# B&R Automation Studio project CleanChemi_SiteManagementSystem (part 4)

#### HA_Find_R.st
```iecst
(* Returns Right index of substring. Negative values are Errors. *)
FUNCTION HA_Find_R
	IF pBuffer = 0 OR pSearch = 0 THEN
		HA_Find_R	 						:= -2;
	ELSE
		Internal.sB							:= brsstrlen(pBuffer);
		Internal.sS							:= brsstrlen(pSearch);
		IF Internal.sB = 0 OR Internal.sB < Internal.sS THEN
		HA_Find_R	 						:= -3;
		END_IF;
	END_IF;
	IF HA_Find_R = 0 THEN
		HA_Find_R							:= -1;
		IF Internal.sS = 0 THEN
			HA_Find_R 						:= 0;
			RETURN;
		ELSE
			FOR Internal.i := 0 TO Internal.sB-Internal.sS DO
				IF brsmemcmp(pBuffer+Internal.i,pSearch,Internal.sS) = 0 THEN
					HA_Find_R 				:= Internal.i+Internal.sS;
					RETURN;
				END_IF;
			END_FOR;
		END_IF;
	END_IF;
END_FUNCTION
```

#### HA_Find_Extract.st
```iecst
(* Negative values are Errors. *)
FUNCTION HA_Find_Extract
	IF pBuffer = 0 OR pSearchL = 0 OR pSearchR = 0 OR pExtractADR = 0 OR pExtractSIZEOF = 0 THEN
		HA_Find_Extract 						:= -2;
	ELSE
		Internal.sB								:= brsstrlen(pBuffer);
		Internal.sSL							:= brsstrlen(pSearchL);
		Internal.sSR							:= brsstrlen(pSearchR);
		IF Internal.sB = 0 OR Internal.sB < (Internal.sSL + Internal.sSR + 1) THEN
			HA_Find_Extract 					:= -3;
		END_IF;
	END_IF;
	IF HA_Find_Extract = 0 THEN
		HA_Find_Extract							:= -1;
		Internal.P1 							:= HA_Find_R(pBuffer,pSearchL);
		IF Internal.P1 >= 0 THEN
			Internal.P2 						:= HA_Find_L(pBuffer+Internal.P1,pSearchR);
			IF Internal.P2 >= 0 THEN
				Internal.Pos 					:= Internal.P1 + pBuffer;
				Internal.Len 					:= DINT_TO_UDINT(Internal.P2);
				brsmemcpy(pExtractADR,ADR(Internal.Pos),4);
				brsmemcpy(pExtractSIZEOF,ADR(Internal.Len),4);
				HA_Find_Extract					:= Internal.P1+Internal.P2+Internal.sSR;
			END_IF;
		END_IF;
	END_IF;
END_FUNCTION
```

### Library Logical/Libraries/API_Login (IEC)

#### Enums.typ
```iecst
TYPE
	LoginState_Enum :
		(
		IDLE_I,
		REQ_AUTH_C,
		REQ_AUTH_W,
		PARSE_AUTH_JSON_C,
		PARSE_AUTH_JSON_W,
		REQ_USER_INFO_W,
		REQ_USER_INFO_C,
		PARSE_USER_INFO_C,
		PARSE_USER_INFO_W,
		CREATE_USER_C,
		CREATE_USER_W,
		SET_PASSWORD_C,
		SET_PASSWORD_W,
		SET_ROLES_W,
		SET_ROLES_C,
		USER_CREATED_SUCCESSS,
		LOGIN_API_ERROR
		);
END_TYPE
```

#### API_Login.fun - Exported functions and function blocks
```iecst
FUNCTION_BLOCK API_Login_FB
	VAR_INPUT
		bExecute : BOOL;
		sUser : STRING[80];
		sPassword : STRING[80];
	END_VAR
	VAR_OUTPUT
		LoginState : LoginState_Enum;
		UserID : STRING[80];
		Password : STRING[80];
		Name : STRING[80];
		Error : BOOL;
		ErrorInfo : STRING[80];
		Done : BOOL;
		Authorization_Bearer : STRING[300];
		ReturnedLastName : STRING[80];
		ReturnedFirstName : STRING[80];
		ReturnedID : UINT;
		ReturnedRole : STRING[80];
	END_VAR
	VAR_IN_OUT
		RequestHeader : httpRequestHeader_t;
		HttpClientRef : httpsClient;
	END_VAR
	VAR
		IdxJSON : DINT;
		GET_UserInfo : GET_UserInfo_FB;
		POST_Login : POST_Login_FB;
		HA_JSON_Parse : HA_JSON_Parse;
		ArUserAssignRole : ArUserAssignRole;
		ArUserSetPassword : ArUserSetPassword;
		JSON_Parsed : ARRAY[0..MAX_JSON_PARSE_PAIR_IDX] OF HA_JSON_Parse_Pair_typ;
		ArUserCreate : ArUserCreate;
	END_VAR
END_FUNCTION_BLOCK

{REDUND_ERROR} FUNCTION_BLOCK POST_Login_FB (*TODO: Add your comment here*) (*$GROUP=User,$CAT=User,$GROUPICON=User.png,$CATICON=User.png*)
	VAR_INPUT
		username : STRING[80];
		password : STRING[80];
		bEnable : BOOL;
		bRequest : BOOL;
	END_VAR
	VAR_OUTPUT
		Phase : UINT;
		Status : {REDUND_UNREPLICABLE} UINT;
		ResponseStatus : {REDUND_UNREPLICABLE} STRING[280];
		Authorization : STRING[200];
		ResponseData : {REDUND_UNREPLICABLE} STRING[2000];
	END_VAR
	VAR_IN_OUT
		HttpClientRef : httpsClient;
		RequestHeader : httpRequestHeader_t;
	END_VAR
	VAR
		Host : {REDUND_UNREPLICABLE} STRING[80];
		ResponseHeader : {REDUND_UNREPLICABLE} httpResponseHeader_t;
		Ressource : {REDUND_UNREPLICABLE} STRING[80];
		sHeader : {REDUND_UNREPLICABLE} STRING[300];
		bEnabled : {REDUND_UNREPLICABLE} BOOL;
		RequestDataJson : {REDUND_UNREPLICABLE} STRING[1000];
	END_VAR
END_FUNCTION_BLOCK

{REDUND_ERROR} FUNCTION_BLOCK GET_UserInfo_FB (*TODO: Add your comment here*) (*$GROUP=User,$CAT=User,$GROUPICON=User.png,$CATICON=User.png*)
	VAR_INPUT
		sAuthorization : STRING[250];
		bEnable : BOOL;
		bRequest : BOOL;
	END_VAR
	VAR_OUTPUT
		Phase : UINT;
		Status : {REDUND_UNREPLICABLE} UINT;
		ResponseStatus : {REDUND_UNREPLICABLE} STRING[280];
		ResponseData : {REDUND_UNREPLICABLE} STRING[2000];
	END_VAR
	VAR_IN_OUT
		HttpClientRef : httpsClient;
		RequestHeader : httpRequestHeader_t;
	END_VAR
	VAR
		Host : {REDUND_UNREPLICABLE} STRING[80];
		ResponseHeader : {REDUND_UNREPLICABLE} httpResponseHeader_t;
		Ressource : {REDUND_UNREPLICABLE} STRING[80];
		sHeader : {REDUND_UNREPLICABLE} STRING[400];
		bEnabled : {REDUND_UNREPLICABLE} BOOL;
		RequestDataJson : {REDUND_UNREPLICABLE} STRING[1000];
	END_VAR
END_FUNCTION_BLOCK
```

#### POST_Login.st
```iecst
(* TODO: Add your comment here *)
FUNCTION_BLOCK POST_Login_FB

	IF bEnable AND NOT bEnabled THEN
		bEnabled	:= TRUE;
		Ressource	:= '/auth/jwt/create/';
		RequestDataJson := CONCAT('{"username":"',username);
		RequestDataJson := CONCAT(	RequestDataJson,'","password":"');
		RequestDataJson := CONCAT(	RequestDataJson,password);
		RequestDataJson := CONCAT(	RequestDataJson,'"}');

		HttpClientRef.method 			:= httpMETHOD_POST;
		HttpClientRef.pUri 				:= ADR(Ressource);
		HttpClientRef.pRequestHeader	:= ADR(RequestHeader);
		HttpClientRef.pRequestData		:= ADR(RequestDataJson);
		HttpClientRef.requestDataLen	:= LEN(RequestDataJson)+2; //According to WireShark there is a /r/n in the packet that is not being accounted for which requires us to add 2 bytes to the length
		HttpClientRef.pResponseHeader	:= ADR(ResponseHeader);
		HttpClientRef.pResponseData 	:= ADR(ResponseData);
		HttpClientRef.responseDataSize	:= SIZEOF(ResponseData);

		RequestHeader.protocol			:= 'HTTP/1.1';
		RequestHeader.host				:= Host;
		RequestHeader.contentType		:= 'application/json';
		RequestHeader.contentLength		:=  LEN(RequestDataJson)+2; //According to WireShark there is a /r/n in the packet that is not being accounted for which requires us to add 2 bytes to the length
		RequestHeader.connection		:= 'keep-alive';
		RequestHeader.rawHeader.dataLen	:= LEN(sHeader);
		RequestHeader.rawHeader.pData	:= ADR(sHeader);

	ELSIF bEnable AND bEnabled THEN
		HttpClientRef.enable	:= TRUE;
		IF bRequest THEN
			HttpClientRef.send	:= TRUE;
		END_IF
	ELSIF NOT bEnable AND bEnabled THEN
		bEnabled	:= FALSE;
		bRequest	:= FALSE;
		HttpClientRef.enable	:= FALSE;
		HttpClientRef.send	:= FALSE;
	END_IF

	HttpClientRef();

	Status := HttpClientRef.status;
	Phase := HttpClientRef.phase;
	ResponseStatus := ResponseHeader.status;

END_FUNCTION_BLOCK
```

#### GET_UserInfo.st
```iecst
(* TODO: Add your comment here *)
FUNCTION_BLOCK GET_UserInfo_FB

	IF bEnable AND NOT bEnabled THEN
		bEnabled	:= TRUE;
		sHeader		:= CONCAT('Authorization: Bearer ',sAuthorization);
		Ressource	:= '/auth/users/me/';

		HttpClientRef.option 			:= httpOPTION_HTTP_11;
		HttpClientRef.method 			:= httpMETHOD_GET;
		HttpClientRef.pUri 				:= ADR(Ressource);
		HttpClientRef.pRequestHeader	:= ADR(RequestHeader);
		HttpClientRef.pRequestData		:= ADR(RequestDataJson);
		HttpClientRef.requestDataLen	:= LEN(RequestDataJson);
		HttpClientRef.pResponseHeader	:= ADR(ResponseHeader);
		HttpClientRef.pResponseData 	:= ADR(ResponseData);
		HttpClientRef.responseDataSize	:= SIZEOF(ResponseData);

		RequestHeader.protocol			:= 'HTTP/1.1';
		RequestHeader.contentType		:= 'application/json';
		RequestHeader.contentLength		:=  LEN(RequestDataJson);
		RequestHeader.connection		:= 'keep-alive';
		RequestHeader.rawHeader.dataLen	:= LEN(sHeader);
		RequestHeader.rawHeader.pData	:= ADR(sHeader);

	ELSIF bEnable AND bEnabled THEN
		HttpClientRef.enable	:= TRUE;
		IF bRequest THEN
			HttpClientRef.send	:= TRUE;
		END_IF
	ELSIF NOT bEnable AND bEnabled THEN
		bEnabled	:= FALSE;
		bRequest	:= FALSE;
		HttpClientRef.enable	:= FALSE;
		HttpClientRef.send	:= FALSE;
	END_IF

	HttpClientRef();

	Status := HttpClientRef.status;
	Phase := HttpClientRef.phase;
	ResponseStatus := ResponseHeader.status;

END_FUNCTION_BLOCK
```

#### API_Login_FB.st
```iecst
(* TODO: Add your comment here *)
FUNCTION_BLOCK API_Login_FB

	IF NOT bExecute THEN
		LoginState := IDLE_I;
	END_IF;

	CASE LoginState OF

		IDLE_I:

			GET_UserInfo.bEnable := FALSE;
			GET_UserInfo.bRequest := FALSE;
			POST_Login.bEnable := FALSE;
			POST_Login.bRequest := FALSE;
			HA_JSON_Parse.Enable := FALSE;
			ArUserSetPassword.Execute := FALSE;
			ArUserCreate.Execute := FALSE;
			brsmemset(ADR(Authorization_Bearer),0,SIZEOF(Authorization_Bearer));
			brsmemset(ADR(JSON_Parsed),0,SIZEOF(JSON_Parsed));
			ErrorInfo := '';

			Done := FALSE;
			Error := FALSE;

			IF bExecute THEN
				LoginState := REQ_AUTH_C;
			END_IF;

		REQ_AUTH_C:

			POST_Login.username := sUser;
			POST_Login.password := sPassword;

			POST_Login.bEnable := TRUE;
			POST_Login.bRequest := TRUE;

			LoginState := REQ_AUTH_W;

		REQ_AUTH_W:

			IF POST_Login.Status = 0 AND POST_Login.ResponseStatus = '200 OK' THEN
				LoginState := PARSE_AUTH_JSON_C;
			ELSIF  POST_Login.Status = 0 AND POST_Login.ResponseStatus = '401 Unauthorized' THEN
				LoginState := LOGIN_API_ERROR;
				ErrorInfo := POST_Login.ResponseStatus;
			ELSIF POST_Login.Status = 0 AND POST_Login.ResponseStatus = '400 Bad Request' THEN
				LoginState := LOGIN_API_ERROR;
				ErrorInfo := POST_Login.ResponseStatus;
			END_IF;

		PARSE_AUTH_JSON_C:

			POST_Login.bEnable := FALSE;
			POST_Login.bRequest := FALSE;
			HA_JSON_Parse.Enable := TRUE;
			HA_JSON_Parse.pBuffer := ADR(POST_Login.ResponseData);
			HA_JSON_Parse.pPairs := ADR(JSON_Parsed);

			LoginState := PARSE_AUTH_JSON_W;

		PARSE_AUTH_JSON_W:

			IF HA_JSON_Parse.Done THEN
				LoginState := REQ_USER_INFO_C;
			END_IF;

		REQ_USER_INFO_C:

			HA_JSON_Parse.Enable := FALSE;

			FOR IdxJSON := 0 TO MAX_JSON_PARSE_PAIR_IDX DO
				IF JSON_Parsed[IdxJSON].Name = 'access' THEN
					brsmemcpy(ADR(Authorization_Bearer),ADR(JSON_Parsed[IdxJSON].Value)+1,LEN(JSON_Parsed[IdxJSON].Value)-2);
					EXIT;
				END_IF;
			END_FOR;

			GET_UserInfo.bEnable := TRUE;
			GET_UserInfo.bRequest := TRUE;
			GET_UserInfo.sAuthorization := Authorization_Bearer;

			LoginState := REQ_USER_INFO_W;

		REQ_USER_INFO_W:

			IF GET_UserInfo.Status = 0 AND GET_UserInfo.ResponseStatus = '200 OK' THEN
				LoginState := PARSE_USER_INFO_C;
			ELSIF GET_UserInfo.Status = 0 AND GET_UserInfo.ResponseStatus = '401 Unauthorized' THEN
				LoginState := LOGIN_API_ERROR;
			END_IF;

		PARSE_USER_INFO_C:

			GET_UserInfo.bEnable := FALSE;
			GET_UserInfo.bRequest := FALSE;
			HA_JSON_Parse.Enable := TRUE;
			HA_JSON_Parse.pBuffer := ADR(GET_UserInfo.ResponseData);
			HA_JSON_Parse.pPairs := ADR(JSON_Parsed);

			LoginState := PARSE_USER_INFO_W;

		PARSE_USER_INFO_W:

			IF HA_JSON_Parse.Done THEN

				FOR IdxJSON := 0 TO MAX_JSON_PARSE_PAIR_IDX DO
					IF JSON_Parsed[IdxJSON].Name = 'role' THEN
						brsmemcpy(ADR(ReturnedRole),ADR(JSON_Parsed[IdxJSON].Value)+1,LEN(JSON_Parsed[IdxJSON].Value)-2);
						EXIT;
					END_IF;
				END_FOR;

				brsmemset(ADR(ReturnedID),0,SIZEOF(ReturnedID));
				FOR IdxJSON := 0 TO MAX_JSON_PARSE_PAIR_IDX DO
					IF JSON_Parsed[IdxJSON].Name = 'id' THEN
						ReturnedID := STRING_TO_USINT(JSON_Parsed[IdxJSON].Value);
						EXIT;
					END_IF;
				END_FOR;

				brsmemset(ADR(ReturnedFirstName),0,SIZEOF(ReturnedFirstName));
				FOR IdxJSON := 0 TO MAX_JSON_PARSE_PAIR_IDX DO
					IF JSON_Parsed[IdxJSON].Name = 'first_name' THEN
						brsmemcpy(ADR(ReturnedFirstName),ADR(JSON_Parsed[IdxJSON].Value)+1,LEN(JSON_Parsed[IdxJSON].Value)-2);
						EXIT;
					END_IF;
				END_FOR;

				brsmemset(ADR(ReturnedLastName),0,SIZEOF(ReturnedLastName));
				FOR IdxJSON := 0 TO MAX_JSON_PARSE_PAIR_IDX DO
					IF JSON_Parsed[IdxJSON].Name = 'last_name' THEN
						brsmemcpy(ADR(ReturnedLastName),ADR(JSON_Parsed[IdxJSON].Value)+1,LEN(JSON_Parsed[IdxJSON].Value)-2);
						EXIT;
					END_IF;
				END_FOR;

				LoginState := CREATE_USER_C;
			END_IF;

		CREATE_USER_C:

			ArUserCreate.Execute := TRUE;
			ArUserCreate.UserName := sUser;

			LoginState := CREATE_USER_W;

		CREATE_USER_W:

			IF ArUserCreate.Done THEN
				LoginState := SET_PASSWORD_C;
			ELSIF ArUserCreate.ErrorID = arUSER_ERR_ALREADY_EXISTS THEN
				LoginState := SET_PASSWORD_C;
			END_IF;

		SET_PASSWORD_C:

			ArUserSetPassword.Execute := TRUE;
			ArUserSetPassword.UserName := sUser;
			ArUserSetPassword.Password := sPassword;

			LoginState := SET_PASSWORD_W;

		SET_PASSWORD_W:

			IF ArUserSetPassword.Done THEN
				LoginState := SET_ROLES_C;
			ELSIF ArUserSetPassword.Error THEN
				CASE ArUserSetPassword.ErrorID OF
					arUSER_ERR_PARAMETER:
						LoginState := LOGIN_API_ERROR;
					arUSER_ERR_DOES_NOT_EXIST:
						LoginState := LOGIN_API_ERROR;
					arUSER_ERR_INTERNAL:
						LoginState := LOGIN_API_ERROR;
				END_CASE;
			END_IF;

		SET_ROLES_C:

			ArUserAssignRole.Execute := TRUE;
			ArUserAssignRole.UserName := sUser;
			ArUserAssignRole.RoleName := ReturnedRole;

			LoginState := SET_ROLES_W;

		SET_ROLES_W:

			IF ArUserAssignRole.Done THEN
				LoginState := USER_CREATED_SUCCESSS;
			ELSIF ArUserAssignRole.Error THEN
				CASE ArUserAssignRole.ErrorID OF
					arUSER_ERR_PARAMETER:

					arUSER_ERR_DOES_NOT_EXIST:
						ErrorInfo := 'User Role Returned from Login API Does NOT Exist on Target System';
						LoginState := LOGIN_API_ERROR;
					arUSER_ERR_ALREADY_EXISTS:
						LoginState := USER_CREATED_SUCCESSS;
					arUSER_ERR_INTERNAL :
						ErrorInfo := 'Unknown Error Occured Setting User Permissions';
						LoginState := LOGIN_API_ERROR;
				END_CASE;
			END_IF;

		USER_CREATED_SUCCESSS:

			Done := TRUE;

		LOGIN_API_ERROR:

			GET_UserInfo.bEnable := FALSE;
			GET_UserInfo.bRequest := FALSE;
			POST_Login.bEnable := FALSE;
			POST_Login.bRequest := FALSE;
			HA_JSON_Parse.Enable := FALSE;
			ArUserSetPassword.Execute := FALSE;
			ArUserCreate.Execute := FALSE;
			ArUserAssignRole.Execute := FALSE;

			Error := TRUE;

	END_CASE;

	GET_UserInfo(HttpClientRef := HttpClientRef, RequestHeader := RequestHeader);
	POST_Login(HttpClientRef := HttpClientRef, RequestHeader := RequestHeader);
	HA_JSON_Parse();
	ArUserSetPassword();
	ArUserCreate();
	ArUserAssignRole();

END_FUNCTION_BLOCK
```

### Library Logical/Libraries/HA_Recipe (IEC)

#### Types.typ - Exported data types
```iecst
TYPE
	Recipe_Definition_typ : 	STRUCT
		MpLink : MpComIdentType;
		VarName : STRING[100];
		pVar : UDINT;
		SizeVar : UDINT;
		pCmpVar : UDINT;
		pDefaultVar : UDINT;
		DeviceName : STRING[50];
		FileName : STRING[255];
	END_STRUCT;
	HA_Recipe_Helper_Internal_typ : 	STRUCT
		MpRecipeRegPar_0 : MpRecipeRegPar;
		MpRecipeXml_0 : MpRecipeXml;
		LastState : HA_RECIPE_HELPER_STATE_ENUM;
		State : HA_RECIPE_HELPER_STATE_ENUM;
		ErrorReset : BOOL;
		CTON_Timeout : CTON;
	END_STRUCT;
	HA_RECIPE_HELPER_STATE_ENUM :
		(
		HA_RH_ST_RESET,
		HA_RH_ST_VALIDATE_INPUTS,
		HA_RH_ST_REG_PAR_W,
		HA_RH_ST_READY,
		HA_RH_ST_SAVE_W,
		HA_RH_ST_LOAD_W,
		HA_RH_ST_AUTO_LOAD_W,
		HA_RH_ST_AUTO_RESET_D,
		HA_RH_ST_AUTO_RESET_C,
		HA_RH_ST_AUTO_RESET_W,
		HA_RH_ST_AUTO_SAVE_W,
		HA_RH_ST_ERROR
		);
END_TYPE
```

#### HA_Recipe.fun - Exported functions and function blocks
```iecst
{REDUND_ERROR} FUNCTION_BLOCK HA_Recipe_Helper (*A helper block for MpRecipe*) (*$GROUP=User,$CAT=User,$GROUPICON=User.png,$CATICON=User.png*)
	VAR_INPUT
		Enable : BOOL;
		Def : Recipe_Definition_typ;
		RemOK : BOOL;
		ErrorReset : BOOL;
		ForceLoad : BOOL;
		ForceSave : BOOL;
		ForceDefaults : BOOL;
	END_VAR
	VAR_OUTPUT
		AutoLoadSuccess : BOOL;
		AutoLoadFailed : BOOL;
		RemLost : BOOL;
		Initialized : BOOL;
		Ready : BOOL;
		Error : BOOL;
	END_VAR
	VAR
		Internal : HA_Recipe_Helper_Internal_typ;
	END_VAR
END_FUNCTION_BLOCK
```

#### HA_Recipe_Helper.st
```iecst
(* A helper block for MpRecipe *)
FUNCTION_BLOCK HA_Recipe_Helper

//Reset in not enabled
	IF NOT Enable THEN
		Internal.State								:= HA_RH_ST_RESET;
	END_IF;

	//Reset Status Flags
	Ready 											:= FALSE;
	Error											:= FALSE;
	AutoLoadSuccess									:= FALSE;
	AutoLoadFailed									:= FALSE;
	RemLost											:= FALSE;

	//Main Case
	CASE Internal.State OF
		HA_RH_ST_RESET:
			Initialized								:= FALSE;
			Internal.ErrorReset 					:= FALSE;
			Internal.MpRecipeXml_0.Load				:= FALSE;
			Internal.MpRecipeXml_0.Save				:= FALSE;
			Internal.State							:= HA_RH_ST_VALIDATE_INPUTS;
		HA_RH_ST_VALIDATE_INPUTS:
			IF Def.pVar = 0 OR Def.SizeVar = 0 OR Def.DeviceName = '' OR Def.FileName = '' OR Def.VarName = '' THEN
				Internal.State						:= HA_RH_ST_ERROR;
			ELSE
				Internal.State						:= HA_RH_ST_REG_PAR_W;
			END_IF;
		HA_RH_ST_REG_PAR_W:
			Internal.CTON_Timeout.IN				:= TRUE;
			Internal.CTON_Timeout.PT				:= T#2s;
			IF Internal.MpRecipeRegPar_0.Error THEN
				Internal.State						:= HA_RH_ST_ERROR;
			ELSIF Internal.CTON_Timeout.Q THEN
				Internal.State						:= HA_RH_ST_ERROR;
			ELSIF Internal.MpRecipeRegPar_0.Active THEN
				IF RemOK THEN
					Internal.State					:= HA_RH_ST_READY;
				ELSE
					RemLost							:= TRUE;
					Internal.MpRecipeXml_0.Load		:= TRUE;
					Internal.State					:= HA_RH_ST_AUTO_LOAD_W;
				END_IF;
			END_IF;
		HA_RH_ST_READY:
			IF ForceLoad THEN
				Internal.MpRecipeXml_0.Load			:= TRUE;
				Internal.State						:= HA_RH_ST_LOAD_W;
			ELSIF ForceDefaults THEN
				IF Def.pDefaultVar <> 0 THEN
					brsmemcpy(Def.pVar,Def.pDefaultVar,Def.SizeVar);
				ELSE
					brsmemset(Def.pVar,0,Def.SizeVar);
				END_IF;
				Internal.MpRecipeXml_0.Save			:= TRUE;
				Internal.State						:= HA_RH_ST_SAVE_W;
			ELSIF ForceSave THEN
				Internal.MpRecipeXml_0.Save			:= TRUE;
				Internal.State						:= HA_RH_ST_SAVE_W;
			ELSIF Def.pCmpVar <> 0 THEN //AutoSave Enabled
				IF brsmemcmp(Def.pCmpVar,Def.pVar,Def.SizeVar) <> 0 THEN //AutoSave On Change
					brsmemcpy(Def.pCmpVar,Def.pVar,Def.SizeVar);
					Internal.MpRecipeXml_0.Save		:= TRUE;
					Internal.State					:= HA_RH_ST_SAVE_W;
				ELSE
					Ready 							:= TRUE;
					Initialized						:= TRUE;
				END_IF;
			ELSE
				Initialized							:= TRUE;
				Ready 								:= TRUE;
			END_IF;
		HA_RH_ST_LOAD_W:
			Internal.CTON_Timeout.IN				:= TRUE;
			Internal.CTON_Timeout.PT				:= T#2s;
			IF (NOT Internal.MpRecipeXml_0.CommandBusy AND Internal.MpRecipeXml_0.Error) OR Internal.CTON_Timeout.Q THEN
				Internal.MpRecipeXml_0.Load			:= FALSE;
				Internal.State						:= HA_RH_ST_ERROR;
			ELSIF (NOT Internal.MpRecipeXml_0.CommandBusy AND Internal.MpRecipeXml_0.CommandDone AND NOT Internal.MpRecipeXml_0.Error) THEN
				Internal.MpRecipeXml_0.Load			:= FALSE;
				Internal.State						:= HA_RH_ST_READY;
			END_IF;
		HA_RH_ST_SAVE_W:
			Internal.CTON_Timeout.IN				:= TRUE;
			Internal.CTON_Timeout.PT				:= T#2s;
			IF (NOT Internal.MpRecipeXml_0.CommandBusy AND Internal.MpRecipeXml_0.Error) OR Internal.CTON_Timeout.Q THEN
				Internal.MpRecipeXml_0.Save			:= FALSE;
				Internal.State						:= HA_RH_ST_ERROR;
			ELSIF (NOT Internal.MpRecipeXml_0.CommandBusy AND Internal.MpRecipeXml_0.CommandDone AND NOT Internal.MpRecipeXml_0.Error) THEN
				Internal.MpRecipeXml_0.Save			:= FALSE;
				Internal.State						:= HA_RH_ST_READY;
			END_IF;
		HA_RH_ST_AUTO_LOAD_W:
			Internal.CTON_Timeout.IN				:= TRUE;
			Internal.CTON_Timeout.PT				:= T#2s;
			IF (NOT Internal.MpRecipeXml_0.CommandBusy AND Internal.MpRecipeXml_0.Error) OR Internal.CTON_Timeout.Q THEN
				AutoLoadFailed						:= TRUE;
				IF Def.pDefaultVar <> 0 THEN
					brsmemcpy(Def.pVar,Def.pDefaultVar,Def.SizeVar);
				ELSE
					brsmemset(Def.pVar,0,Def.SizeVar);
				END_IF;
				Internal.MpRecipeXml_0.Load			:= FALSE;
				Internal.State						:= HA_RH_ST_AUTO_RESET_D;
			ELSIF (NOT Internal.MpRecipeXml_0.CommandBusy AND Internal.MpRecipeXml_0.CommandDone AND NOT Internal.MpRecipeXml_0.Error) THEN
				AutoLoadSuccess						:= TRUE;
				Internal.MpRecipeXml_0.Load			:= FALSE;
				Internal.State						:= HA_RH_ST_READY;
			END_IF;
		HA_RH_ST_AUTO_RESET_D:
			Internal.State							:= HA_RH_ST_AUTO_RESET_C;
		HA_RH_ST_AUTO_RESET_C:
			Internal.ErrorReset						:= TRUE;
			Internal.State							:= HA_RH_ST_AUTO_RESET_W;
		HA_RH_ST_AUTO_RESET_W:
			Internal.CTON_Timeout.IN				:= TRUE;
			Internal.CTON_Timeout.PT				:= T#2s;
			IF Internal.CTON_Timeout.Q THEN
				Internal.ErrorReset					:= FALSE;
				Internal.State						:= HA_RH_ST_ERROR;
			ELSIF NOT Internal.MpRecipeXml_0.Error THEN
				Internal.ErrorReset					:= FALSE;
				Internal.MpRecipeXml_0.Save			:= TRUE;
				Internal.State						:= HA_RH_ST_AUTO_SAVE_W;
			END_IF;
		HA_RH_ST_AUTO_SAVE_W:
			Internal.CTON_Timeout.IN				:= TRUE;
			Internal.CTON_Timeout.PT				:= T#2s;
			IF (NOT Internal.MpRecipeXml_0.CommandBusy AND Internal.MpRecipeXml_0.Error) OR Internal.CTON_Timeout.Q THEN
				Internal.MpRecipeXml_0.Save			:= FALSE;
				Internal.State						:= HA_RH_ST_ERROR;
			ELSIF (NOT Internal.MpRecipeXml_0.CommandBusy AND Internal.MpRecipeXml_0.CommandDone AND NOT Internal.MpRecipeXml_0.Error) THEN
				Internal.MpRecipeXml_0.Save			:= FALSE;
				Internal.State						:= HA_RH_ST_READY;
			END_IF;
		HA_RH_ST_ERROR:
			Error									:= TRUE;
			IF ErrorReset THEN
				Internal.State						:= HA_RH_ST_RESET;
			END_IF;
	END_CASE;

	//Reset Commands
	ForceDefaults 									:= FALSE;
	ForceLoad 										:= FALSE;
	ForceSave 										:= FALSE;

	//Reset Timeout On State Change
	IF Internal.LastState <> Internal.State OR Internal.State = HA_RH_ST_RESET THEN
		Internal.LastState 							:= Internal.State;
		Internal.CTON_Timeout.IN					:= FALSE;
	END_IF;

	//FB Calls
	Internal.CTON_Timeout();
	Internal.MpRecipeRegPar_0(MpLink := ADR(Def.MpLink), Enable := Enable, ErrorReset := (ErrorReset OR Internal.ErrorReset), PVName := ADR(Def.VarName), Category := ADR(Def.VarName));
	Internal.MpRecipeXml_0(MpLink := ADR(Def.MpLink), Enable := Enable, ErrorReset := (ErrorReset OR Internal.ErrorReset), DeviceName := ADR(Def.DeviceName), FileName := ADR(Def.FileName), Category := ADR(Def.VarName));

END_FUNCTION_BLOCK
```

- Alarms.mpalarmxcore_temp (not shown)

### Library Logical/Libraries/HA_Sim (IEC)

#### Types.typ - Exported data types
```iecst
TYPE
	HA_Sim_Actuator_TF_Internal_typ : 	STRUCT
		Active : BOOL;
		OldDampingRatio : REAL;
		OldNaturalFreq : REAL;
		OldFullStrokeValue : REAL;
		MTBasicsTransferFcn_0 : MTBasicsTransferFcn;
	END_STRUCT;
	HA_Sim_Actuator_Lin_Internal_typ : 	STRUCT
		Active : BOOL;
		OldTimePos : REAL;
		OldTimeNeg : REAL;
		MTBasicsLimiter_0 : MTBasicsLimiter;
	END_STRUCT;
END_TYPE
```

#### HA_Sim.fun - Exported functions and function blocks
```iecst
{REDUND_ERROR} FUNCTION_BLOCK HA_Sim_Actuator_Lin (* *) (*$GROUP=User,$CAT=User,$GROUPICON=User.png,$CATICON=User.png*)
	VAR_INPUT
		Enable : BOOL;
		Actuate : BOOL;
		FullStrokeValue : REAL;
		FeedbackTol : REAL;
		TimeNeg : REAL;
		TimePos : REAL;
	END_VAR
	VAR_OUTPUT
		Position : REAL;
		AtFalsePosition : BOOL;
		AtTruePosition : BOOL;
		Error : BOOL;
	END_VAR
	VAR
		Internal : HA_Sim_Actuator_Lin_Internal_typ;
	END_VAR
END_FUNCTION_BLOCK

{REDUND_ERROR} FUNCTION_BLOCK HA_Sim_Actuator_TF (* *) (*$GROUP=User,$CAT=User,$GROUPICON=User.png,$CATICON=User.png*)
	VAR_INPUT
		Enable : BOOL;
		Actuate : BOOL;
		ClampValueToEnds : BOOL;
		FullStrokeValue : REAL;
		FeedbackTol : REAL;
		NaturalFreq : REAL;
		DampingRatio : REAL;
	END_VAR
	VAR_OUTPUT
		Position : REAL;
		AtFalsePosition : BOOL;
		AtTruePosition : BOOL;
		Error : BOOL;
	END_VAR
	VAR
		Internal : HA_Sim_Actuator_TF_Internal_typ;
	END_VAR
END_FUNCTION_BLOCK
```

#### HA_Sim_Actuator_TF.st
```iecst
FUNCTION_BLOCK HA_Sim_Actuator_TF

	IF Enable THEN
		IF NOT Internal.Active OR (Internal.Active AND (Internal.OldNaturalFreq <> NaturalFreq OR Internal.OldDampingRatio <> DampingRatio OR Internal.OldFullStrokeValue <> FullStrokeValue)) THEN
			Internal.MTBasicsTransferFcn_0.Numerator[0] 	:= FullStrokeValue*NaturalFreq**2;
			Internal.MTBasicsTransferFcn_0.Denominator[0] 	:= NaturalFreq**2;
			Internal.MTBasicsTransferFcn_0.Denominator[1] 	:= 2*DampingRatio*NaturalFreq;
			Internal.MTBasicsTransferFcn_0.Denominator[2] 	:= 1;
			Internal.OldNaturalFreq							:= NaturalFreq;
			Internal.OldDampingRatio						:= DampingRatio;
			Internal.OldFullStrokeValue						:= FullStrokeValue;
			IF Internal.Active THEN
				Internal.MTBasicsTransferFcn_0.Update		:= TRUE;
			END_IF;
			Internal.Active 								:= TRUE;
		END_IF;

		IF Actuate THEN
			Internal.MTBasicsTransferFcn_0.In				:= 1.0;
		ELSE
			Internal.MTBasicsTransferFcn_0.In				:= 0.0;
		END_IF;

		Position 											:= Internal.MTBasicsTransferFcn_0.Out;
		IF ClampValueToEnds THEN
			IF Internal.MTBasicsTransferFcn_0.Out > FullStrokeValue THEN
				Position 									:= FullStrokeValue;
			ELSIF Internal.MTBasicsTransferFcn_0.Out < 0 THEN
				Position 									:= 0.0;
			END_IF;
		END_IF;

		AtFalsePosition										:= ABS(Position) <= FeedbackTol;
		AtTruePosition										:= ABS(Position-FullStrokeValue) <= FeedbackTol;
		Internal.MTBasicsTransferFcn_0.Enable				:= TRUE;
	ELSE
		Position 											:= 0.0;
		AtFalsePosition 									:= FALSE;
		AtTruePosition 										:= FALSE;
		Internal.Active 									:= FALSE;
		Internal.MTBasicsTransferFcn_0.Enable				:= FALSE;
		Internal.MTBasicsTransferFcn_0.In					:= 0.0;
		Internal.OldNaturalFreq								:= 0.0;
		Internal.OldDampingRatio							:= 0.0;
		Internal.OldFullStrokeValue							:= 0.0;
	END_IF;

	Internal.MTBasicsTransferFcn_0();
	Internal.MTBasicsTransferFcn_0.Update 					:= FALSE;
	Error 													:= Internal.MTBasicsTransferFcn_0.Error;

END_FUNCTION_BLOCK
```

#### HA_Sim_Actuator_Lin.st
```iecst
FUNCTION_BLOCK HA_Sim_Actuator_Lin

	IF Enable THEN
		IF NOT Internal.Active OR (Internal.Active AND (Internal.OldTimeNeg <> TimeNeg OR Internal.OldTimePos <> TimePos)) THEN
			IF TimeNeg <= 0 THEN
				Internal.MTBasicsLimiter_0.MaxNegSlewRate	:= 0;
			ELSE
				Internal.MTBasicsLimiter_0.MaxNegSlewRate	:= 1.0/TimeNeg;
			END_IF;
			IF TimePos <= 0 THEN
				Internal.MTBasicsLimiter_0.MaxPosSlewRate	:= 0;
			ELSE
				Internal.MTBasicsLimiter_0.MaxPosSlewRate	:= 1.0/TimePos;
			END_IF;
			Internal.OldTimeNeg 							:= TimeNeg;
			Internal.OldTimePos 							:= TimePos;
			IF Internal.Active THEN
				Internal.MTBasicsLimiter_0.Update			:= TRUE;
			END_IF;
			Internal.Active 								:= TRUE;
		END_IF;

		IF Actuate THEN
			Internal.MTBasicsLimiter_0.In					:= 1.0;
		ELSE
			Internal.MTBasicsLimiter_0.In					:= 0.0;
		END_IF;

		Position 											:= Internal.MTBasicsLimiter_0.Out*FullStrokeValue;

		AtFalsePosition										:= ABS(Position) <= FeedbackTol;
		AtTruePosition										:= ABS(Position-FullStrokeValue) <= FeedbackTol;
		Internal.MTBasicsLimiter_0.Enable					:= TRUE;
	ELSE
		Position 											:= 0.0;
		AtFalsePosition 									:= FALSE;
		AtTruePosition 										:= FALSE;
		Internal.Active 									:= FALSE;
		Internal.MTBasicsLimiter_0.Enable					:= FALSE;
		Internal.MTBasicsLimiter_0.In						:= 0.0;
		Internal.OldTimeNeg									:= 0.0;
		Internal.OldTimePos									:= 0.0;
	END_IF;

	Internal.MTBasicsLimiter_0();
	Internal.MTBasicsLimiter_0.Update 						:= FALSE;
	Error 													:= Internal.MTBasicsLimiter_0.Error;

END_FUNCTION_BLOCK
```

### Package Logical/modbusTCP - Programs

### Library Logical/modbusTCP/MbusTCP (ANSIC, version 2.00.0)
Depends on: astcp, standard, astime, AsBrStr, AsARCfg, sys_lib, AsIecCon

#### Types.typ - Exported data types
```iecst
TYPE
	step_enum :
		( (*local state machine*)
		INIT,
		GET_IP,
		WAIT_SERVER,
		OPEN_PORT,
		SET_LINGER,
		SET_NODELAY,
		WAIT_CONNECTION,
		WAIT_REQUEST,
		SEND_ANSWER,
		CREATE_REQUEST,
		SEND_REQUEST,
		WAIT_ANSWER,
		CLOSE_PORT,
		WAIT,
		ERROR
		);
	step_sub_enum :
		(
		SUB_WAIT,
		SUB_SEND,
		SUB_CLOSE_MASTER
		);
	receive_buff_typ : 	STRUCT  (*Receive data buffer*)
		byte : ARRAY[0..500]OF USINT; (*Received data*)
	END_STRUCT;
	t_master_request : 	STRUCT
		transaction_id : UINT;
		protocol_id : UINT;
		length : UINT;
		unit : USINT;
		function_code : USINT;
		quantity : UINT;
	END_STRUCT;
	t_read_request : 	STRUCT
		starting_addr : UINT;
		quantity : UINT;
	END_STRUCT;
	t_single_write_request : 	STRUCT
		starting_addr : UINT;
		value : UINT;
	END_STRUCT;
	t_multiple_write_request : 	STRUCT
		starting_addr : UINT;
		quantity : UINT;
		byte_nr : UINT;
	END_STRUCT;
	master_info_typ : 	STRUCT
		ident : UDINT;
		port : UINT;
		ip_addr : ARRAY[0..17]OF USINT; (*Client IP address*)
		timeout_timer : TON; (*Timer to determine when connection times out*)
		disconnect : BOOL; (*Flag to disconnect this client if it times out.*)
	END_STRUCT;
	modbus_master_action_enable_typ : 	STRUCT
		cyclic : BOOL;
		single : BOOL;
	END_STRUCT;
	modbus_master_action_param_typ : 	STRUCT
		unit : USINT;
		type : USINT;
		start_addr : UINT;
		quantity : UINT;
		p_pv : UDINT;
		timer : UDINT;
	END_STRUCT;
	modbus_master_cfg_typ : 	STRUCT
		action_enable : ARRAY[0..MASTER_MAX_ACTION_INDEX]OF modbus_master_action_enable_typ;
		action_param : ARRAY[0..MASTER_MAX_ACTION_INDEX]OF modbus_master_action_param_typ;
	END_STRUCT;
	modbus_master_internal_typ : 	STRUCT  (*Internal master variables*)
		step : UINT; (*Internal state in a state machine*)
		cycle_time : UINT;
		time_old : TIME;
		tcp_open : TcpOpen; (*TcpOpen FUB from AsTCP*)
		tcp_ioctl : TcpIoctl; (*TcpIoctl FUB from AsTCP*)
		tcp_client : TcpClient; (*TcpClient FUB from AsTCP*)
		tcp_send : TcpSend; (*TcpSend FUB from AsTCP*)
		tcp_receive : TcpRecv; (*TcpRecv FUB from AsTCP*)
		tcp_close : TcpClose; (*TcpClose FUB from AsTCP*)
		tcp_ip : CfgGetIPAddr;
		linger_opt : tcpLINGER_typ; (*TcpIoctl linger options*)
		last_req : USINT; (*Last request*)
		receive_timer : UDINT; (*Receive timer*)
		send_timer : ARRAY[0..MASTER_MAX_ACTION_INDEX]OF UDINT; (*Send timer*)
		send_buff : ARRAY[0..500]OF USINT; (*Send buffer*)
		receive_buff : ARRAY[0..500]OF USINT; (*Receive buffer*)
		transaction_id : UINT; (*Transaction ID*)
		wrong_message : UDINT; (*Wrong message counter*)
	END_STRUCT;
	modbus_slave_cfg_typ : 	STRUCT
		p_discrete_inputs : ARRAY[0..SLAVE_MAX_REGISTER_INDEX]OF UDINT;
		p_coils : ARRAY[0..SLAVE_MAX_REGISTER_INDEX]OF UDINT;
		p_input_registers : ARRAY[0..SLAVE_MAX_REGISTER_INDEX]OF UDINT;
		p_holding_registers : ARRAY[0..SLAVE_MAX_REGISTER_INDEX]OF UDINT;
	END_STRUCT;
	modbus_slave_internal_typ : 	STRUCT  (*Internal slave variables*)
		step : UINT; (*Internal state in a state machine*)
		substep : step_sub_enum; (*Internal substate in a state machine*)
		i : USINT; (*Loop counter*)
		master_nr : USINT; (*Client ID*)
		master_last : USINT;
		master_info : ARRAY[0..SLAVE_MAX_CONNECTION_INDEX]OF master_info_typ; (*Client info*)
		master_addr : ARRAY[0..17]OF USINT; (*Client IP address*)
		tcp_open : TcpOpen; (*TcpOpen FUB from AsTCP*)
		tcp_ioctl : TcpIoctl; (*TcpIoctl FUB from AsTCP*)
		tcp_server : TcpServer; (*TcpServer FUB from AsTCP*)
		tcp_send : TcpSend; (*TcpSend FUB from AsTCP*)
		tcp_receive : ARRAY[0..SLAVE_MAX_CONNECTION_INDEX]OF TcpRecv; (*TcpRecv FUB from AsTCP*)
		tcp_close : TcpClose; (*TcpClose FUB from AsTCP*)
		tcp_ip : CfgGetIPAddr;
		linger_opt : tcpLINGER_typ; (*TcpIoctl linger options*)
		send_buff : ARRAY[0..500]OF USINT; (*Send buffer*)
		send_byte : UINT;
		receive_buff : ARRAY[0..SLAVE_MAX_CONNECTION_INDEX]OF receive_buff_typ; (*Receive buffers for clients*)
	END_STRUCT;
END_TYPE
```

#### Variables.var
```iecst
(*----------------------------------------------------------------------------------------------------------------------------------------------------------------------*)
(*General configuration*)
VAR CONSTANT
	LOG_LINE_NUM : USINT := 50; (*Number of log entries*)
	LOG_LINE_LEN : USINT := 100; (*Size of one log entry*)
	LLN : USINT := LOG_LINE_NUM; (*Shorter variable name for indexing logger. String was too long*)
	LLL : USINT := LOG_LINE_LEN; (*Shorter variable name for indexing logger. String was too long*)
	SLAVE_MAX_CONNECTION_NUM : USINT := 3; (*Maximum number of slave connections to master*)
	SLAVE_MAX_REGISTER_NUM : UINT := 256; (*Maximum number of slave registers*)
	MASTER_MAX_ACTION_NUM : UINT := 140; (*Maximum number of master actions*)
END_VAR
(*----------------------------------------------------------------------------------------------------------------------------------------------------------------------*)
(*Modbus functions*)
VAR CONSTANT
	READ_COILS : USINT := 16#01;
	READ_DISCRETE_INPUTS : USINT := 16#02;
	READ_HOLDING_REGISTERS : USINT := 16#03;
	READ_INPUT_REGISTERS : USINT := 16#04;
	WRITE_SINGLE_COIL : USINT := 16#05;
	WRITE_SINGLE_REGISTER : USINT := 16#06;
	WRITE_MULTIPLE_COILS : USINT := 16#0F;
	WRITE_MULTIPLE_REGISTERS : USINT := 16#10;
	ON : UINT := 16#FF00;
	OFF : UINT := 16#0000;
END_VAR
(*----------------------------------------------------------------------------------------------------------------------------------------------------------------------*)
(*Error numbers*)
VAR CONSTANT
	ERROR_CRITICAL : UINT := 50000; (* COM: Critical error, disable and re-enable FUB *)
	ERROR_MESSAGE_SIZE : UINT := 50001; (* COM: Frame message is TO short *)
	ERROR_MESSAGE_FORMAT : UINT := 50002; (* COM: Message format is incorrect *)
	ERROR_REC_BUF_EXCEEDED : UINT := 50003; (* COM: Receive buffer exceeded maximum configured size *)
	ERROR_ADR_EMPTY : UINT := 50004; (* COM: Variable address is empty *)
	ERROR_QUANTITY : UINT := 50006; (* COM: Quantity is higher than the Modbus limit (125 for analog/2000 for digital) *)
	ERROR_TOO_MANY_MASTERS : UINT := 50100; (* SLV: More than MAX_MASTER are trying TO connect *)
	ERROR_ADR_EXCEEDED : UINT := 50101; (* SLV: Address exceeded maximum configured size *)
	ERROR_LENGTH_EXCEEDED : UINT := 50102; (* SLV: Address+Size exceeded maximum configured size or modbus limit (125/2000) *)
	ERROR_FUNCTION_CODE : UINT := 50103; (* SLV: Function code is not supported *)
	ERROR_MASTER_TIMED_OUT : UINT := 50104; (* SLV: The master did not send a request for a certain TIME *)
	ERROR_CFG_MASTERS : UINT := 50110; (* SLV: Configuration error in num masters *)
	ERROR_BAD_SLAVE_DATA : UINT := 50200; (* MAS: Bad data received from slave *)
	ERROR_SLAVE_DATA_TOO_SHORT : UINT := 50201; (* MAS: Data received from slave too short *)
	ERROR_SLAVE_DATA_TOO_LONG : UINT := 50202; (* MAS: Data received from slave too long *)
	ERROR_TIMEOUT_REQ : UINT := 50210; (* MAS: A slave request timed out *)
	ERROR_TIMEOUT_CONNECT : UINT := 50211; (* MAS: Connection request timed out *)
	ERROR_DEVICE_ERR : UINT := 50300; (* MAS: Invalid Ethernet device *)
END_VAR
(**)
VAR CONSTANT
	ERROR_MOD_FUNCTION : UINT := 16#01; (* Modbus error: wrong function code *)
	ERROR_MOD_ADR : UINT := 16#02; (* Modbus error: wrong address *)
	ERROR_MOD_VALUE : UINT := 16#03; (* Modbus error: wrong value *)
END_VAR
(*----------------------------------------------------------------------------------------------------------------------------------------------------------------------*)
(*Log book messages*)
VAR CONSTANT
	TYP_REQUEST : USINT := 0;
	TYP_RESPONSE : USINT := 1;
END_VAR
(*----------------------------------------------------------------------------------------------------------------------------------------------------------------------*)
(*Other constants*)
VAR CONSTANT
	SLAVE_MAX_CONNECTION_INDEX : USINT := SLAVE_MAX_CONNECTION_NUM-1;
	SLAVE_MAX_REGISTER_INDEX : UINT := SLAVE_MAX_REGISTER_NUM-1;
	MASTER_MAX_ACTION_INDEX : USINT := MASTER_MAX_ACTION_NUM-1;
	MODBUS_TCP_PORT : UINT := 502;
	MODBUS_MAX_REG : UINT := 125; (* Maximum number of modbus registers for one request *)
	DISABLE : UINT := 65534;
	BUSY : UINT := 65535;
	RECEIVE_TIMEOUT : UINT := 5000;
	DEBUG_LEVEL : USINT := 2;
END_VAR
```

#### MbusTCP.fun - Exported functions and function blocks
```iecst
FUNCTION_BLOCK MBslave (*ModbusTCP slave implementation*)
	VAR_INPUT
		enable : BOOL; (*Enable execution*)
		device : UDINT; (*Ethernet device string*)
		port : UINT; (*Port number of the slave (default 502)*)
		p_cfg : REFERENCE TO modbus_slave_cfg_typ; (*Pointer to data*)
		p_log : UDINT; (*Pointer to logger array*)
		master_timeout : UDINT; (*Master has to send at least one request within this time (ms).  (0 to disable)*)
	END_VAR
	VAR_OUTPUT
		my_ip : STRING[20]; (*Device IP address*)
		status : UINT; (*Execution status: ERR_OK, ERR_FUB_ENABLE_FALSE, ERR_FUB_BUSY, 0xXXXX = see help*)
		last_error : UINT; (*Error number of data request from the client*)
	END_VAR
	VAR
		internal : modbus_slave_internal_typ; (*Internal variables and FUBs*)
	END_VAR
END_FUNCTION_BLOCK

FUNCTION_BLOCK MBmaster (*ModbusTCP master implementation*)
	VAR_INPUT
		enable : BOOL; (*Enable execution*)
		device : UDINT; (*Ethernet device string*)
		port : UINT; (*Port number of the slave (default 502)*)
		slave_ip_addr : STRING[18]; (*IP address of the slave*)
		p_cfg : REFERENCE TO modbus_master_cfg_typ; (*Pointer to configuration data*)
		p_log : UDINT; (*Pointer to logger array*)
	END_VAR
	VAR_OUTPUT
		last_error : UINT; (*Error number of data response from the slave*)
		my_ip : STRING[20]; (*Device IP address*)
		status : UINT; (*Execution status: ERR_OK, ERR_FUB_ENABLE_FALSE, ERR_FUB_BUSY, 0xXXXX = see help*)
	END_VAR
	VAR
		internal : modbus_master_internal_typ; (*Internal variables and FUBs*)
	END_VAR
END_FUNCTION_BLOCK
```

#### MBmaster.c - Master
```c
// -------------------------------------------------------------------------------------------------
// Library: MbusTCP
// Author: Stephan Stricker
// Created: October 29, 2022
// -------------------------------------------------------------------------------------------------

#include <bur/plctypes.h>
#ifdef __cplusplus
	extern "C"
	{
#endif
#include "MbusTCP.h"
#ifdef __cplusplus
	};
#endif

// -------------------------------------------------------------------------------------------------
// Local functions
// -------------------------------------------------------------------------------------------------
UINT create_request_to_slave (struct modbus_master_cfg_typ* config, USINT req_nr, USINT* send_buff, UINT size_buf, UINT transaction_id, UDINT p_log);
UINT analyze_answer_from_slave (struct modbus_master_cfg_typ* config, USINT req_nr, USINT* receive_buff, UINT transaction_id, UDINT p_log);

UINT MySwapUINT(UINT data);
INT MySwapINT(INT data);
void NewLogEntry(STRING message[LOG_LINE_LEN], UDINT p_log);
void MessageLog(USINT type, USINT function_code, UINT start_addr, UINT length, UDINT p_log);

// -------------------------------------------------------------------------------------------------
// Master function block
// -------------------------------------------------------------------------------------------------
void MBmaster(struct MBmaster* inst)
{
	USINT	x;
	USINT	receive_status;
	TIME 	time_new;

	// Increase cycle timers when connected
	if(inst->internal.step > WAIT_CONNECTION)
	{
		time_new = clock_ms();
		inst->internal.cycle_time = time_new - inst->internal.time_old;

		// Make sure cycle time has a value
		if(inst->internal.cycle_time != 0 && inst->internal.time_old != 0)
		{
			for(x=0;x<sizeof((*(inst->p_cfg)).action_param)/sizeof((*(inst->p_cfg)).action_param[0]);x++)
				inst->internal.send_timer[x] += inst->internal.cycle_time;
		}
		inst->internal.time_old = time_new;
	}
	switch(inst->internal.step)
	{
		// ------------------------------------------------------------------------------------------
		// Assign buffers and port
		case INIT:
			inst->internal.tcp_send.pData 		= (UDINT)inst->internal.send_buff;
			inst->internal.tcp_receive.pData	= (UDINT)inst->internal.receive_buff;
			inst->internal.tcp_receive.datamax	= sizeof(inst->internal.receive_buff);
			if(inst->port == 0) inst->port = MODBUS_TCP_PORT;
			inst->internal.step = DISABLE;
		// ------------------------------------------------------------------------------------------
		// Wait for function block enable
		case DISABLE:
			if(inst->enable)
			{
				inst->internal.step = GET_IP;
				NewLogEntry("Validating own ip...", inst->p_log);
			}
		break;
		// ------------------------------------------------------------------------------------------
		// Read own IP address
		case GET_IP:
			if(inst->enable)
			{
				inst->internal.tcp_ip.enable 	= 1;
				inst->internal.tcp_ip.pDevice 	= (UDINT)inst->device;
				inst->internal.tcp_ip.pIPAddr 	= (UDINT)inst->my_ip;
				inst->internal.tcp_ip.Len 		= 18;
				CfgGetIPAddr(&inst->internal.tcp_ip);
				inst->status = inst->internal.tcp_ip.status;
				// --------------------------------------------------------------------------------------
				// Success
				if (inst->internal.tcp_ip.status == 0)
				{
					if(brsstrcmp((UDINT)inst->my_ip, (UDINT)"0.0.0.0") == 0) break;
					inst->internal.step = OPEN_PORT;
				}
				else if(inst->internal.tcp_ip.status == cfgERR_DEVICE_NOT_EXIST)
				{
					NewLogEntry("ERR: Invalid ethernet device", inst->p_log);
					inst->status 		= ERROR_DEVICE_ERR;
					inst->internal.step = ERROR;
				}
				else if(inst->internal.tcp_ip.status != BUSY) inst->internal.step = ERROR;
			}
			else inst->internal.step = CLOSE_PORT;
		break;
		// ------------------------------------------------------------------------------------------
		// Open ethernet port
		case OPEN_PORT:
			if(inst->enable)
			{
				inst->internal.tcp_open.options = tcpOPT_REUSEADDR;
				inst->internal.tcp_open.enable 	= 1;
				TcpOpen(&inst->internal.tcp_open);
				// --------------------------------------------------------------------------------------
				// Success
				if (inst->internal.tcp_open.status == 0)
				{
					NewLogEntry("Open port successful", inst->p_log);
					inst->internal.tcp_client.enable	= 1;
					inst->internal.tcp_client.ident		= inst->internal.tcp_open.ident;
					inst->internal.tcp_client.pServer	= (UDINT)inst->slave_ip_addr;
					inst->internal.tcp_client.portserv	= inst->port;
					inst->internal.tcp_send.ident		= inst->internal.tcp_open.ident;
					inst->internal.tcp_receive.ident	= inst->internal.tcp_open.ident;
					NewLogEntry("Trying to connect...", inst->p_log);
					inst->internal.step = WAIT_CONNECTION;
				}
				else if(inst->internal.tcp_open.status != BUSY)
				{
					NewLogEntry("ERR: open port failed", inst->p_log);
					inst->internal.step = ERROR;
				}
				inst->status = inst->internal.tcp_open.status;
			}
			else inst->internal.step = CLOSE_PORT;
			inst->status = inst->internal.tcp_open.status;
		break;
		// ------------------------------------------------------------------------------------------
		// Open ethernet port
		case WAIT_CONNECTION:
			if(inst->enable)
			{
				inst->internal.tcp_client.enable = 1;
				TcpClient(&inst->internal.tcp_client);
				inst->status = inst->internal.tcp_client.status;
				// ----------------------------------------------------------------------------------
				// Success
				if(inst->internal.tcp_client.status == 0)
				{
					NewLogEntry("Connected", inst->p_log);
					inst->internal.step = CREATE_REQUEST;
				}
				else if(inst->internal.tcp_client.status == tcpERR_INVALID)
				{
					NewLogEntry("ERR: Cant find slave", inst->p_log);
					inst->status = ERROR_TIMEOUT_CONNECT;
					inst->internal.step = CLOSE_PORT;
				}
				else if(inst->internal.tcp_client.status != BUSY)
				{
					NewLogEntry("ERR: Could not establish connection", inst->p_log);
					inst->status = ERROR_TIMEOUT_CONNECT;
					inst->internal.step = ERROR;
				}
			}
			else inst->internal.step = CLOSE_PORT;
		break;
		// ------------------------------------------------------------------------------------------
		// Create new requests
		case CREATE_REQUEST:
			if(inst->enable)
			{
				UINT tmp_req = inst->internal.last_req;
				// ----------------------------------------------------------------------------------
				// Find next request
				do
				{
					// ----------------------------------------------------------------------------------
					// Switch to next action, roll over
					inst->internal.last_req++;
					if(((*(inst->p_cfg)).action_param[inst->internal.last_req].p_pv == 0) || (inst->internal.last_req >= sizeof((*(inst->p_cfg)).action_param)/sizeof((*(inst->p_cfg)).action_param[0]))) inst->internal.last_req=0;
					// ----------------------------------------------------------------------------------
					// Execute action when set to single or timer is expired
					if (((*(inst->p_cfg)).action_enable[inst->internal.last_req].single) ||
						((inst->internal.send_timer[inst->internal.last_req] >= (*(inst->p_cfg)).action_param[inst->internal.last_req].timer) && ((*(inst->p_cfg)).action_enable[inst->internal.last_req].cyclic)))
					{
						if(((*(inst->p_cfg)).action_param[inst->internal.last_req].p_pv) != 0)
						{
							USINT function_code = (*(inst->p_cfg)).action_param[inst->internal.last_req].type;
							UINT quantity = (*(inst->p_cfg)).action_param[inst->internal.last_req].quantity;
							if ((function_code	== READ_COILS || function_code	== READ_DISCRETE_INPUTS || function_code == WRITE_MULTIPLE_COILS) && quantity > MODBUS_MAX_REG*2*8)
							{
								NewLogEntry("ERR: Max length exceeded", inst->p_log);
								inst->status = ERROR_QUANTITY;
								inst->last_error = ERROR_QUANTITY;
								(*(inst->p_cfg)).action_enable[inst->internal.last_req].single = 0;
							}
							else if ((function_code	== READ_HOLDING_REGISTERS || function_code	== READ_INPUT_REGISTERS || function_code == WRITE_MULTIPLE_REGISTERS) && quantity > MODBUS_MAX_REG)
							{
								NewLogEntry("ERR: Max length exceeded", inst->p_log);
								inst->status = ERROR_QUANTITY;
								inst->last_error = ERROR_QUANTITY;
								(*(inst->p_cfg)).action_enable[inst->internal.last_req].single = 0;
							}
							else
							{
								inst->internal.step = SEND_REQUEST;
								inst->internal.transaction_id++;
								inst->internal.tcp_send.datalen = create_request_to_slave((modbus_master_cfg_typ*)(inst->p_cfg), inst->internal.last_req, inst->internal.send_buff, sizeof(inst->internal.send_buff), inst->internal.transaction_id, inst->p_log);
							}
							inst->internal.send_timer[inst->internal.last_req] = 0;
						}
						else // Variable address is empty
						{
						NewLogEntry("ERR: Empty variable ADR", inst->p_log);
						inst->status 		= ERROR_ADR_EMPTY;
						inst->internal.step = ERROR;
						}
						break;
					}
					if(inst->internal.last_req == tmp_req) break;
				}
				while(1);
			}
			else inst->internal.step = CLOSE_PORT;
		break;
		// ------------------------------------------------------------------------------------------
		// Create new requests
		case SEND_REQUEST:
			if(inst->enable)
			{
				inst->internal.tcp_send.enable = 1;
				TcpSend(&inst->internal.tcp_send);
				// ----------------------------------------------------------------------------------
				// Success
				if(inst->internal.tcp_send.status == 0)
				{
					inst->internal.receive_timer = 0;
					inst->internal.step = WAIT_ANSWER;
				}
				else if(((inst->internal.tcp_send.status != BUSY) 				&&
					     (inst->internal.tcp_send.status != tcpERR_WOULDBLOCK)	&&
					     (inst->internal.tcp_send.status != tcpERR_SENTLEN))    ||
						 (inst->internal.tcp_send.status == tcpERR_NOT_CONNECTED))	inst->internal.step = CLOSE_PORT;
			}
			else inst->internal.step = CLOSE_PORT;
			inst->status = inst->internal.tcp_send.status;
		break;
		// ------------------------------------------------------------------------------------------
		// Wait for answer
		case WAIT_ANSWER:
			if(inst->enable)
			{
				inst->internal.tcp_receive.enable = 1;
				TcpRecv(&inst->internal.tcp_receive);
				// ----------------------------------------------------------------------------------
				// Success
				if(inst->internal.tcp_receive.status == 0)
				{
					if(inst->internal.tcp_receive.recvlen != 0)
					{
						if((inst->internal.tcp_receive.recvlen > 8) && (inst->internal.tcp_receive.recvlen < sizeof(inst->internal.receive_buff)))
						{
							receive_status = analyze_answer_from_slave((modbus_master_cfg_typ*)(inst->p_cfg), inst->internal.last_req, inst->internal.receive_buff, inst->internal.transaction_id, inst->p_log);
							if(receive_status) inst->last_error = ERROR_BAD_SLAVE_DATA;
						}
						else if(inst->internal.tcp_receive.recvlen >= sizeof(inst->internal.receive_buff))
						{
							NewLogEntry("ERR: Data received too long", inst->p_log);
							receive_status = 1;
							inst->last_error = ERROR_SLAVE_DATA_TOO_LONG;
						}
						else
						{
							NewLogEntry("ERR: Data received too short", inst->p_log);
							receive_status = 1;
							inst->last_error = ERROR_SLAVE_DATA_TOO_SHORT;
						}
						if(receive_status) 	inst->internal.wrong_message ++;
						(*(inst->p_cfg)).action_enable[inst->internal.last_req].single = 0;
						inst->internal.step = CREATE_REQUEST;
					}
					else inst->internal.step = CLOSE_PORT;
				}
				else if((inst->internal.tcp_receive.status != BUSY) &&
					    (inst->internal.tcp_receive.status != tcpERR_NO_DATA)) inst->internal.step = CLOSE_PORT;
				// ----------------------------------------------------------------------------------
				// See if request timed out
				inst->internal.receive_timer += inst->internal.cycle_time;
				if (inst->internal.receive_timer >= RECEIVE_TIMEOUT)
				{
					NewLogEntry("ERR: Request timed out", inst->p_log);
					inst->status = ERROR_TIMEOUT_REQ;
					inst->last_error = ERROR_TIMEOUT_REQ;
					inst->internal.step = CREATE_REQUEST;
					break;
				}
			}
			else inst->internal.step = CLOSE_PORT;
			if(inst->internal.tcp_receive.status != tcpERR_NO_DATA)	inst->status = inst->internal.tcp_receive.status;
			else													inst->status = 0;
		break;
		// ------------------------------------------------------------------------------------------
		// Close connection
		case CLOSE_PORT:
			inst->internal.tcp_close.enable 	= 1;
			inst->internal.tcp_close.ident		= inst->internal.tcp_open.ident;
			inst->internal.tcp_close.how 		= 0;
			TcpClose(&inst->internal.tcp_close);
			// --------------------------------------------------------------------------------------
			// Success
			if(inst->internal.tcp_close.status == 0)
			{
				NewLogEntry("Port closed", inst->p_log);
				inst->internal.send_timer[0] = 0;
				inst->internal.step = WAIT;
			}
			else if(inst->internal.tcp_close.status == tcpERR_INVALID_IDENT)
			{
				inst->internal.step = ERROR;
			}
			inst->status = inst->internal.tcp_close.status;
		break;
		// ------------------------------------------------------------------------------------------
		// Wait before reopen port
		case WAIT:
			inst->internal.tcp_open.enable = 0;
			TcpOpen(&inst->internal.tcp_open);
			inst->internal.tcp_client.enable = 0;
			TcpClient(&inst->internal.tcp_client);

			inst->internal.send_timer[0] += inst->internal.cycle_time;
			if (inst->internal.send_timer[0] > 1000) inst->internal.step = OPEN_PORT;
		break;
		// ------------------------------------------------------------------------------------------
		// Error state
		case ERROR:
			if (inst->status < 50000) inst->status = ERROR_CRITICAL;
			if (inst->enable == 0) inst->internal.step = DISABLE;
		break;
	}
}

// -------------------------------------------------------------------------------------------------
// Create new request to slave
// -------------------------------------------------------------------------------------------------
UINT create_request_to_slave(struct modbus_master_cfg_typ* config, USINT req_nr, USINT* send_buff, UINT size_buf, UINT transaction_id, UDINT p_log)
{
	UINT	uint_var;
	INT		int_var;
	INT		value;
	UINT	data_len, i;

	// Error message for undefined function code
	brsmemset((UDINT)send_buff, 0, size_buf);
	// Transaction id: 2 byte
	uint_var = MySwapUINT(transaction_id);
	brsmemcpy((UDINT)&send_buff[0], (UDINT)&uint_var, sizeof(uint_var));
	// Protocol id: 2 byte
	uint_var = 0;
	brsmemcpy((UDINT)&send_buff[2], (UDINT)&uint_var, sizeof(uint_var));
	// Length: 2 byte
	// Unit: 1 byte
	send_buff[6] = (*config).action_param[req_nr].unit;
	switch((*config).action_param[req_nr].type)
	{
		case READ_COILS:
			// Function code: 1 byte
			send_buff[7] = READ_COILS;
			// Starting address: 2 byte
			uint_var = MySwapUINT((*config).action_param[req_nr].start_addr);
			brsmemcpy((UDINT)&send_buff[8], (UDINT)&uint_var, sizeof(uint_var));
			// Coils number: 2 byte
			uint_var = MySwapUINT((*config).action_param[req_nr].quantity);
			brsmemcpy((UDINT)&send_buff[10], (UDINT)&uint_var, sizeof(uint_var));
			// Data len
			data_len = 6;
			break;
		case READ_DISCRETE_INPUTS:
			// Function code: 1 byte
			send_buff[7] = READ_DISCRETE_INPUTS;
			// Starting address: 2 byte
			uint_var = MySwapUINT((*config).action_param[req_nr].start_addr);
			brsmemcpy((UDINT)&send_buff[8], (UDINT)&uint_var, sizeof(uint_var));
			// Inputs number: 2 byte
			uint_var = MySwapUINT((*config).action_param[req_nr].quantity);
			brsmemcpy((UDINT)&send_buff[10], (UDINT)&uint_var, sizeof(uint_var));
			// Data length
			data_len = 6;
			break;
		case READ_HOLDING_REGISTERS:
			// Function code: 1 byte
			send_buff[7] = READ_HOLDING_REGISTERS;
			// Starting address: 2 byte
			uint_var = MySwapUINT((*config).action_param[req_nr].start_addr);
			brsmemcpy((UDINT)&send_buff[8], (UDINT)&uint_var, sizeof(uint_var));
			// Holding registers number: 2 byte
			uint_var = MySwapUINT((*config).action_param[req_nr].quantity);
			brsmemcpy((UDINT)&send_buff[10], (UDINT)&uint_var, sizeof(uint_var));
			// Data length
			data_len = 6;
			break;
		case READ_INPUT_REGISTERS:
			// Function code: 1 byte
			send_buff[7] = READ_INPUT_REGISTERS;
			// Starting address: 2 byte
			uint_var = MySwapUINT((*config).action_param[req_nr].start_addr);
			brsmemcpy((UDINT)&send_buff[8], (UDINT)&uint_var, sizeof(uint_var));
			// Input registers number: 2 byte
			uint_var = MySwapUINT((*config).action_param[req_nr].quantity);
			brsmemcpy((UDINT)&send_buff[10], (UDINT)&uint_var, sizeof(uint_var));
			// Data length
			data_len = 6;
			break;
		case WRITE_SINGLE_COIL:
			// Function code: 1 byte
			send_buff[7] = WRITE_SINGLE_COIL;
			// Starting address: 2 byte
			uint_var = MySwapUINT((*config).action_param[req_nr].start_addr);
			brsmemcpy((UDINT)&send_buff[8], (UDINT)&uint_var, sizeof(uint_var));
			// Value: 2 byte
			if(*((BOOL*)((*config).action_param[req_nr].p_pv)))	value = ON;
			else												value = OFF;
			int_var = MySwapINT(value);
			brsmemcpy((UDINT)&send_buff[10], (UDINT)&int_var, sizeof(int_var));
			// Data length
			data_len = 6;
			break;
		case WRITE_SINGLE_REGISTER:
			// Function code: 1 byte
			send_buff[7] = WRITE_SINGLE_REGISTER;
			// Starting address: 2 byte
			uint_var = MySwapUINT((*config).action_param[req_nr].start_addr);
			brsmemcpy((UDINT)&send_buff[8], (UDINT)&uint_var, sizeof(uint_var));
			// Value: 2 byte
			value = *((INT*)((*config).action_param[req_nr].p_pv));
			int_var = MySwapINT(value);
			brsmemcpy((UDINT)&send_buff[10], (UDINT)&int_var, sizeof(int_var));
			// Data length
			data_len = 6;
			break;
		case WRITE_MULTIPLE_COILS:
			// Function code: 1 byte
			send_buff[7] = WRITE_MULTIPLE_COILS;
			// Starting address: 2 byte
			uint_var = MySwapUINT((*config).action_param[req_nr].start_addr);
			brsmemcpy((UDINT)&send_buff[8], (UDINT)&uint_var, sizeof(uint_var));
			// Quantity: 2 byte
			uint_var = MySwapUINT((*config).action_param[req_nr].quantity);
			brsmemcpy((UDINT)&send_buff[10], (UDINT)&uint_var, sizeof(uint_var));
			// Byte count: 1 byte
			if( (*config).action_param[req_nr].quantity % 8)	send_buff[12] = ((*config).action_param[req_nr].quantity / 8) + 1;
			else												send_buff[12] = (*config).action_param[req_nr].quantity / 8;
			// Coil value: x byte
			for(i = 0; i < (*config).action_param[req_nr].quantity; i++)
			{
				if(	((BOOL*)((*config).action_param[req_nr].p_pv))[i])
					send_buff[13 + (i/8)] = send_buff[13 + (i/8)] | (USINT)(0x01 << (i%8));
				else
					send_buff[13 + (i/8)] = send_buff[13 + (i/8)] & (USINT)~(0x01 << (i%8));
			}
			// Data length
			data_len = 7 + send_buff[12];
			break;

		case WRITE_MULTIPLE_REGISTERS:
			// Function code: 1 byte
			send_buff[7] = WRITE_MULTIPLE_REGISTERS;
			// Starting address: 2 byte
			uint_var = MySwapUINT((*config).action_param[req_nr].start_addr);
			brsmemcpy((UDINT)&send_buff[8], (UDINT)&uint_var, sizeof(uint_var));
			// Quantity: 2 byte
			uint_var = MySwapUINT((*config).action_param[req_nr].quantity);
			brsmemcpy((UDINT)&send_buff[10], (UDINT)&uint_var, sizeof(uint_var));
			// Byte count: 1 byte
			send_buff[12] = (*config).action_param[req_nr].quantity * 2;
			// Coil value: x byte
			for(i = 0; i < (*config).action_param[req_nr].quantity; i++)
			{
				value = ((INT*)((*config).action_param[req_nr].p_pv))[i];
				int_var = MySwapINT(value);
				brsmemcpy((UDINT)&send_buff[13 + (i*2)], (UDINT)&int_var, sizeof(int_var));
			}
			// Data length
			data_len = 7 + send_buff[12];
			break;

		default:
			// Unsupported function code
			NewLogEntry("ERR: Client function code", p_log);
			break;
	}
	// Create log entry
	MessageLog (TYP_REQUEST, (*config).action_param[req_nr].type, (*config).action_param[req_nr].start_addr, (*config).action_param[req_nr].quantity, p_log);

	// Length: 2 byte
	uint_var = MySwapUINT(data_len);
	brsmemcpy((UDINT)&send_buff[4], (UDINT)&uint_var, sizeof(uint_var));
	return 6 + data_len;
}

// -------------------------------------------------------------------------------------------------
// Analyse response from slave
// -------------------------------------------------------------------------------------------------
UINT analyze_answer_from_slave(struct modbus_master_cfg_typ* config,USINT req_nr, USINT* receive_buff, UINT transaction_id, UDINT p_log)
{
	INT		int_var;
	UINT	uint_var, receive_tr_id, protocol_id, length;
	UINT	function_code, quantity, i;

	// Transaction id: 2 byte
	brsmemcpy((UDINT)&uint_var, (UDINT)&receive_buff[0], sizeof(uint_var));
	receive_tr_id	= MySwapUINT(uint_var);
	// Protocol id: 2 byte
	brsmemcpy((UDINT)&uint_var, (UDINT)&receive_buff[2], sizeof(uint_var));
	protocol_id		= MySwapUINT(uint_var);
	// Length: 2 byte
	brsmemcpy((UDINT)&uint_var, (UDINT)&receive_buff[4], sizeof(uint_var));
	length 			= MySwapUINT(uint_var);
	// Function code: 1 byte
	function_code	= receive_buff[7];

	if((receive_tr_id 	== transaction_id)	&&
	   (protocol_id		== 0)				&&
	   (length			> 0)				&&
	   (function_code	< 0x80))
	{
		switch(function_code)
		{
			case READ_COILS:
				// Quantity: 1 byte
				quantity = (*config).action_param[req_nr].quantity;
				// Coil value: x byte
				for(i = 0; i < quantity; i++)
				{
					if (receive_buff[9 + (i/8)] & (USINT)(0x01 << (i%8))) 	((BOOL*)((*config).action_param[req_nr].p_pv))[i] = 1;
					else													((BOOL*)((*config).action_param[req_nr].p_pv))[i] = 0;
				}
				break;

			case READ_DISCRETE_INPUTS:
				// Quantity: 1 byte
				quantity = (*config).action_param[req_nr].quantity;
				// Coil value: x byte
				for(i = 0; i < quantity; i++)
				{
					if (receive_buff[9 + (i/8)] & (USINT)(0x01 << (i%8)))	((BOOL*)((*config).action_param[req_nr].p_pv))[i] = 1;
					else													((BOOL*)((*config).action_param[req_nr].p_pv))[i] = 0;
				}
				break;

			case READ_HOLDING_REGISTERS:
				// Quantity: 1 byte
				quantity = receive_buff[8] / 2;
				// Coil value: x byte
				for(i = 0; i < quantity; i++)
				{
					brsmemcpy((UDINT)&int_var, (UDINT)&receive_buff[9 + (i*2)], sizeof(int_var));
					((INT*)((*config).action_param[req_nr].p_pv))[i] = MySwapINT(int_var);
				}
				break;

			case READ_INPUT_REGISTERS:
				// Quantity: 1 byte
				quantity = receive_buff[8] / 2;
				// Coil value: x byte
				for(i = 0; i < quantity; i++)
				{
					brsmemcpy((UDINT)&int_var, (UDINT)&receive_buff[9 + (i*2)], sizeof(int_var));
					((INT*)((*config).action_param[req_nr].p_pv))[i] = MySwapINT(int_var);
				}
				break;

			default:
				// Unsupported function code
				if ((function_code > WRITE_SINGLE_REGISTER) && ((function_code != WRITE_MULTIPLE_COILS) && (function_code != WRITE_MULTIPLE_REGISTERS)))
					NewLogEntry("ERR: Server function code", p_log);
				break;
		}
		// Create log entry
		MessageLog (TYP_RESPONSE, function_code, 0, 0, p_log);
	}
	// Generate error on function exception from slave
	else if(function_code >= 0x80)
	{
		function_code -= 0x80;
		switch(receive_buff[8])
			{
				case 1: NewLogEntry("ERR: Server->Bad function", p_log); break;
				case 2: NewLogEntry("ERR: Server->Data address", p_log); break;
				case 3: NewLogEntry("ERR: Server->Data value", p_log); break;
				case 4: NewLogEntry("ERR: Server->Device failure", p_log); break;
				case 5: NewLogEntry("ERR: Server->Exception ack", p_log); break;
				case 6: NewLogEntry("ERR: Server->Slave busy", p_log); break;
				case 10: NewLogEntry("ERR: Server->Path unavailable", p_log); break;
				default: NewLogEntry("ERR: Server->unknown", p_log); break;
			}
		return 1;
	}
	else
	{
		NewLogEntry("ERR: Bad slave message", p_log);
		return 1;
	}
	return 0;
}
```
